(* CODESYS project codesys-syslog-library-history
   Author: John te Bokkel
   Company: PowerCore Engineering
   CompiledLibraryCompatibilityVersion: CODESYS V3.5 SP16
   DefaultNamespace: Syslog
   Description: Library project to implement RFC 5424 The Syslog Protocol
   DocFormat: reStructuredText
   LanguageModelAttribute: qualified-access-only
   Placeholder: CODESYS_SYSLOG
   Title: Code-Syslog
   Version: 0.1.0.0

Project tree, tasks and I/O mapping:
  libraries: CAA Types Extern, 3.5.17.0 (CAA Technical Workgroup); CAA FB Factory, 3.5.17.0 (CAA Technical Workgroup); Common Behaviour Model, 3.5.17.0 (3S - Smart Software Solutions GmbH); StringUtils, * (System); Code-Syslog Interfaces, * (PowerCore Engineering); SysTimeRtc, 3.5.17.0 (System); Element Collections, 3.5.17.0 (3S - Smart Software Solutions GmbH); CAA File, 3.5.17.0 (CAA Technical Workgroup); Net Base Services, 3.5.17.0 (3S - Smart Software Solutions GmbH); CmpIecTask, 3.5.17.0 (System); CmpCrypto, 3.5.17.0 (System); Standard, 3.5.18.0 (System)
  code-syslog/
  oscat-basic/
    function BIT_COUNT [ST]
    function D_TRUNC [ST]
    function FRACT [ST]
    function RDM [ST]
    function T_PLC_MS [ST]
  Handlers/
    Rotator/
    function block SyslogFileHandler [ST]: Dispatch, p_FlushNow, p_LogSeverity, prvFileSetup, prvFlush, prvProcessQueue, Run
    function block SyslogHandlerBase [ST]: Dispatch, p_LogSeverity, Run
    function block SyslogRotatingFileHandler [ST]: DoRollover, Rotate, RotationFilename, ShouldRollover
    function block SyslogRotatingFileHandlerBase [ST]: Run
    function block SyslogUdpHandler [ST]: prvInit, prvProcessQueue, prvSetupConnection, Run
  Syslog Msg Collection/
    function block IDataSyslogMsgElement [ST]
    interface ISyslogMsgElement: SyslogMsgValue
    function block SyslogMsgElement [ST]: ElementCompareTo, ElementEquals, ElementHashCode, prvInstInit, SyslogMsgValue
    function block SyslogMsgElementFactory [ST]: Create, prvInstCount, prvInstPoolExtendsFactor, prvInstSize
  function block SyslogLogger [ST]: FB_Init, Alert, Critical, Debug, Emergency, Error, Information, Notice, Warning, GetAppName, GetFacility, GetHostname, GetProcId, GetVersion, RegisterHandler, SetAppName, SetFacility, SetHostname, SetProcId, UnregisterHandler, prvBuildSyslogMessage, prvDispatch, prvTimestamp
  function Escape_ParamValue [ST]
  function Make_Priority [ST]
  function Make_SdParam2 [ST]
  function Make_SdParam [ST]
  function Make_SdParamSb [ST]
  function RandomEmpherialPort [ST]
  SafeLog/
    function SyslogAlert [ST]
    function SyslogCritical [ST]
    function SyslogDebug [ST]
    function SyslogEmergency [ST]
    function SyslogError [ST]
    function SyslogInfo [ST]
    function SyslogNotice [ST]
    function SyslogWarning [ST]
  function Sanitize_Msg [ST]
  function Sanitize_PrintUsAscii [ST]
  function Sanitize_SdName [ST]
  function StrucDataMsg [ST]
  function UtcTimestamp [ST]
  function UtcTimestampFromSystimeDate [ST]
  global variables Constants
*)

// Constants
{attribute 'qualified_only'}
//{attribute 'conditionalshow'}
//{attribute 'conditionalshow' := 'SomeText'}
//{attribute 'hide'}
VAR_GLOBAL CONSTANT
	gc_uiMaxHandlers : UINT := 5; /// Max number of registered log handlers
END_VAR

// Handlers/SyslogRotatingFileHandlerBase/DoRollover
/// Perform the rollover
/// :returns: TRUE when complete
{warning 'Add method implementation '}
METHOD PROTECTED DoRollover : BOOL
VAR_INPUT
END_VAR

// Handlers/SyslogRotatingFileHandlerBase/Rotate
/// When rotating, rotate the current log.
/// 
/// This should manage the file handle for the current log file. (ie. close it and reopen)
{warning 'Add method implementation '}
METHOD PROTECTED Rotate : BOOL
VAR_INPUT
	(* The source filename. This is normally the base filename, eg ``test.log``*)
	source	: STRING(255);
	(* The destination filename. This is normally what the source is rotated to, eg ``test.log.1``*)
	dest	: STRING(255);
END_VAR

// Handlers/SyslogRotatingFileHandlerBase/RotationFilename
/// Transformation file naming method.
/// 
/// default_name will be ``sFullFilename.#``
{warning 'Add method implementation '}
METHOD PROTECTED RotationFilename : CAA.FILENAME
VAR_INPUT
	default_name : CAA.FILENAME;
END_VAR

// Handlers/SyslogRotatingFileHandlerBase/ShouldRollover
{warning 'Add method implementation '}
/// Determine if we should rollover for this message. This needs to return in one call.
/// This method needs to look at the next message to be written to determine if rollover should occur.
METHOD PROTECTED ShouldRollover : BOOL
VAR_INPUT
END_VAR

// oscat-basic/BIT_COUNT
FUNCTION BIT_COUNT : INT
VAR_INPUT
	IN : DWORD;
END_VAR


(*
version 1.1	10 sep 2007
programmer 	hugo
tested by		tobias

BIT_COUNT counts the amount True of bits in a dword.
for exabple: bit_count(3) returns 2 because two bits (bits 0 and 1) are true and all others are false. 

*)

WHILE in > 0 DO
	IF in.0 THEN Bit_Count := Bit_Count + 1; END_IF;
	in := SHR(in,1);
END_WHILE;



(* revision history
5.7.2007	rev 1.0		original version

10.9.2007	rev 1.1		hm
	changed algorithm for better performace
	the execution time has reduced by a factor of 5
	deleted unused variable temp
*)

END_FUNCTION

// oscat-basic/D_TRUNC
FUNCTION D_TRUNC : DINT
VAR_INPUT
	X : REAL;
END_VAR

(*
version 1.2	10. mar. 2009
programmer 	hugo
tested by		oscat

d_trunc truncates a real to a dint 1.5 will be 1 and -1.5 will be -1
d_trunc is necessary because many systems do not offer a trunc to a dint
also real_to_dint will not deliver the same result on different systems

*)

D_TRUNC := REAL_TO_DINT(X);
IF X > 0.0 THEN
	IF DINT_TO_REAL(D_TRUNC) > X THEN D_TRUNC := D_TRUNC - 1; END_IF;
ELSE
	IF DINT_TO_REAL(D_TRUNC) < X THEN D_TRUNC := D_TRUNC + 1; END_IF;
END_IF;


(* for systems that support a dint truncation this routine can be replaced by trunc() *)


(* revision history
hm	21. mar. 2008	rev 1.0
	original version

hm	31. oct. 2008	rev 1.1
	optimized performance

hm	10. mar. 2009	rev 1.2
	real constants updated to new systax using dot
*)

END_FUNCTION

// oscat-basic/FRACT
/// this function returns the fraction of a real number
/// fract(3.14) = 0.14
FUNCTION FRACT : REAL
VAR_INPUT
	x : REAL;
END_VAR


(*
version 1.3	10. mar. 2009
programmer 	hugo
tested by		tobias

this function returns the fraction of a real number
fract(3.14) = 0.14

*)

IF ABS(x) < 2.0E9 THEN
	FRACT := x - DINT_TO_REAL(D_TRUNC(x));
ELSE
	FRACT := 0.0;
END_IF;

(* revision history
hm	4. aug 2006	rev 1.0
	original version

hm	11. mar 2008	rev 1.1
	added dint_to_real for compatibility reasons
	now returns 0 for number > 2e9
	changed input to x

hm	21. mar. 2008	rev 1.2
	use D_trunc instead of TRUNC for compatibility reasons

hm	10. mar. 2009	rev 1.3
	real constants updated to new systax using dot

*)

END_FUNCTION

// oscat-basic/RDM
(*this function calculates a pseudo random number
to generate the number it reads the sps timer and calculates a random number between 0 and 1:
in order to use rdm more then once within one sps cycle it need to be called with different seed numbers LAST.
*)
FUNCTION RDM : REAL
VAR_INPUT
	last : REAL;
END_VAR
VAR
	tn : DWORD;
	tc : INT;
END_VAR
VAR CONSTANT
	E : REAL := 	2.71828182845904523536028747135266249;		(* Euler constant e *)
END_VAR

(*
version 1.9	10. mar. 2009
programmer 	hugo
tested by		tobias

this function calculates a pseudo random number
to generate the number it reads the sps timer and calculates a random number between 0 and 1:
in order to use rdm more then once within one sps cycle it need to be called with different seed numbers LAST.

*)

tn := T_PLC_MS();
tc := BIT_COUNT(tn);
tn.31 := tn.2;
tn.30 := tn.5;
tn.29 := tn.4;
tn.28 := tn.1;
tn.27 := tn.0;
tn.26 := tn.7;
tn.25 := tn.6;
tn.24 := tn.3;
tn := ROL(tn,BIT_COUNT(tn)) OR 16#80000001;
tn := tn MOD 71474513 + INT_TO_DWORD(tc + 77);
RDM := FRACT(DWORD_TO_REAL(tn) / 10000000.0 * (E - LIMIT(0.0,last,1.0)));


(*
pt := ADR(temp);
pt^ := (T_PLC_MS() AND 16#007FFFFF) OR 16#3D000000;
RDM := fract(modR(temp*e+pi1, PI1-last) + modR(temp*PI1+e + last,e-last));
*)

(* revision history
hm		16. jan 2007		rev 1.0
	original version

hm		11. nov 2007		rev 1.1
	changed time() into t_plc_ms()

hm		20. nov 2007		rev 1.2
	changed code of temp calculation to avoid overflow in modr due to resuclt would not fit DINT for high timeer values

hm		5. jan 2008		rev 1.3
	changed calculation of temp to avoid problem with high values of t_plc_ms

hm		2. feb 2008		rev 1.4
	changed algorithm to avoind non iec functions and guarantee more randomness

hm	10. mar. 2008		rev 1.5
	make sure last will be between 0 and 1 to avoid invalid results

hm	16. mar. 2008		rev 1.6
	added conversion for tc to avoid warnings under codesys 3.0

hm	18. may. 2008		rev 1.7
	changed constant E to E1

hm	18. oct. 2008		rev 1.8
	using math constants

hm	10. mar. 2009		rev 1.9
	real constants updated to new systax using dot

*)

END_FUNCTION

// oscat-basic/T_PLC_MS
FUNCTION T_PLC_MS : DWORD
VAR CONSTANT
	debug : BOOL := 0;
	N : INT := 0;
	offset : DWORD := 0;
END_VAR
VAR
	tx : TIME;
END_VAR

(*
version 1.2	16. nov 2008
programmer 	hugo
tested by	oscat

T_PLC_MS reads the internal PLC timer and return the time, it has the advantage to be able to set a debug mode 
and speed up the counter to test the plc timer overrun which occurs every 50 days respectively 25 days at siemens S7
this routine also allows to correct the behavior of s7 where the internal plc counter will not count all 32 bits.

*)

tx := TIME();
T_PLC_MS := TIME_TO_DWORD(Tx);
(* hier muss die korrektur für step7 stattfinden
plctime muss den vollen wertebereich von time ausnutzen:
wenn bei step7 time -24tage bis plus 24 tage ist dann muss der timer auch beim überlauf auf -24tage springen 
und auf keinen fall auf 0 !!!!
für siemens muss ein weiterer fb im main eingebunden werden der sicherstellt das alle 32 bits durchgezählt werden.
es kann nur ein fb sein den er muss sich das oberste (32te) bit merken.
oder etwa spring s7 bei überlauf auf -24 tage????? dann wäre keine korrektur nötig.
*)
IF debug THEN
	T_PLC_MS := (SHL(T_PLC_MS,N) OR SHL(DWORD#1,N)-1) + OFFSET;
END_IF;

(* revision history
hm	14.9.2007	rev 1.0
	original version

hm	12. nov 2007	rev 1.1
	added temporaray variable tx because some compilers could not handle time() as an argument

hm	16. nov. 2008	rev 1.2
	initialized constants with 0 for compatibility reasons
*)

END_FUNCTION

// SyslogLogger
FUNCTION_BLOCK SyslogLogger IMPLEMENTS SyslogItfs.ISyslogLogger, SyslogItfs.ISyslogLoggerConfig
VAR_INPUT
END_VAR
VAR_OUTPUT
END_VAR
VAR
	_hostname : SyslogItfs.HOSTNAME := SyslogItfs.Constants.gc_sNILVALUE;
	_appName : SyslogItfs.APP_NAME := SyslogItfs.Constants.gc_sNILVALUE;
	_procId : SyslogItfs.PROC_ID := SyslogItfs.Constants.gc_sNILVALUE;
	_facility : SyslogItfs.SyslogFacility := SyslogItfs.SyslogFacility.USER;
	regHandler : ARRAY [0..c_iMaxHandler] OF SyslogItfs.ISyslogHandler;
	version : SyslogItfs.SYSLOG_VERSION := c_sVersion;
	ixHandler : INT;
END_VAR
VAR CONSTANT
	c_iMaxHandler : INT := UINT_TO_INT(Constants.gc_uiMaxHandlers) - 1;
	c_sVersion : STRING(2) := '1';
END_VAR

FOR ixHandler := 0 TO c_iMaxHandler BY 1 DO
	IF regHandler[ixHandler] <> CAA.gc_hINVALID THEN
		regHandler[ixHandler].Run();
	END_IF
END_FOR

//FB_Init is always available implicitly and it is used primarily for initialization.
//The return value is not evaluated. For a specific influence, you can also declare the
//methods explicitly and provide additional code there with the standard initialization
//code. You can evaluate the return value.
METHOD FB_Init: BOOL
VAR_INPUT
    bInitRetains: BOOL; // TRUE: the retain variables are initialized (reset warm / reset cold)
    bInCopyCode: BOOL;  // TRUE: the instance will be copied to the copy code afterward (online change)   
	hostname : SyslogItfs.HOSTNAME;
	appName : SyslogItfs.APP_NAME;
	procId : SyslogItfs.PROC_ID;
	facility : SyslogItfs.SyslogFacility;
	handler : SyslogItfs.ISyslogHandler;
END_VAR
THIS^._hostname := hostname;
THIS^._appName := appName;
THIS^._procId := procId;
THIS^._facility := facility;

THIS^.RegisterHandler(handler);
END_METHOD

METHOD Alert : BOOL
VAR_INPUT
	msgId	: SyslogItfs.MSG_ID;
	msg	: SyslogItfs.MSG;
END_VAR
THIS^.prvDispatch(SyslogItfs.SyslogSeverity.ALERT, ADR(msgId), ADR(msg));
END_METHOD

METHOD Critical : BOOL
VAR_INPUT
	msgId	: SyslogItfs.MSG_ID;
	msg	: SyslogItfs.MSG;
END_VAR
THIS^.prvDispatch(SyslogItfs.SyslogSeverity.CRITICAL, ADR(msgId), ADR(msg));
END_METHOD

METHOD Debug : BOOL
VAR_INPUT
	msgId	: SyslogItfs.MSG_ID;
	msg	: SyslogItfs.MSG;
END_VAR
THIS^.prvDispatch(SyslogItfs.SyslogSeverity.DEBUG, ADR(msgId), ADR(msg));
END_METHOD

METHOD Emergency : BOOL
VAR_INPUT
	msgId	: SyslogItfs.MSG_ID;
	msg	: SyslogItfs.MSG;
END_VAR
THIS^.prvDispatch(SyslogItfs.SyslogSeverity.EMERGENCY, ADR(msgId), ADR(msg));
END_METHOD


METHOD Error : BOOL
VAR_INPUT
	msgId	: SyslogItfs.MSG_ID;
	msg	: SyslogItfs.MSG;
END_VAR
THIS^.prvDispatch(SyslogItfs.SyslogSeverity.ERROR, ADR(msgId), ADR(msg));
END_METHOD


METHOD Information : BOOL
VAR_INPUT
	msgId	: SyslogItfs.MSG_ID;
	msg	: SyslogItfs.MSG;
END_VAR
THIS^.prvDispatch(SyslogItfs.SyslogSeverity.INFORMATION, ADR(msgId), ADR(msg));
END_METHOD


METHOD Notice : BOOL
VAR_INPUT
	msgId	: SyslogItfs.MSG_ID;
	msg	: SyslogItfs.MSG;
END_VAR
THIS^.prvDispatch(SyslogItfs.SyslogSeverity.NOTICE, ADR(msgId), ADR(msg));
END_METHOD


METHOD Warning : BOOL
VAR_INPUT
	msgId	: SyslogItfs.MSG_ID;
	msg	: SyslogItfs.MSG;
END_VAR
THIS^.prvDispatch(SyslogItfs.SyslogSeverity.WARNING, ADR(msgId), ADR(msg));
END_METHOD

METHOD GetAppName : SyslogItfs.APP_NAME
GetAppName := THIS^._appName;
END_METHOD

METHOD GetFacility : SyslogItfs.SyslogFacility
GetFacility := THIS^._facility;
END_METHOD

METHOD GetHostname : SyslogItfs.HOSTNAME
GetHostname := THIS^._hostname;
END_METHOD

METHOD GetProcId : SyslogItfs.PROC_ID
GetProcId := THIS^._procId;
END_METHOD

METHOD GetVersion : SyslogItfs.SYSLOG_VERSION
GetVersion := THIS^.version;
END_METHOD

/// Register Syslog Handler
/// :returns: TRUE if successfully added
METHOD RegisterHandler : BOOL
VAR_INPUT
	handler : SyslogItfs.ISyslogHandler;
END_VAR
VAR
	xDup : BOOL;
	ix : INT;
	ixOpen : INT;
END_VAR
IF handler <> CAA.gc_hINVALID THEN
	xDup := FALSE;
	ixOpen := -1;
	// We need to check the whole array for dups
	FOR ix := 0 TO c_iMaxHandler BY 1 DO
		xDup S= THIS^.regHandler[ix] = handler;
		IF ixOpen = -1 AND_THEN THIS^.regHandler[ix] = CAA.gc_hINVALID THEN
			ixOpen := ix;
		END_IF
	END_FOR
	
	IF NOT xDup THEN
		IF ixOpen >= 0 AND ixOpen <= c_iMaxHandler THEN
			THIS^.regHandler[ixOpen] := handler;
			RegisterHandler := TRUE;
		END_IF
	END_IF
END_IF
END_METHOD

(* Set App-Name According to RFC5424 Section 6.2.5*)
/// :returns: FALSE if we ended up with an empty/null string otherwise TRUE
METHOD SetAppName : BOOL
VAR_INPUT
	sAppName	: SyslogItfs.APP_NAME;
END_VAR
SetAppName := TRUE;
THIS^._appName := sAppName;

Sanitize_PrintUsAscii(ADR(THIS^._appName));
// Make sure we have a legal name after sanitizing it
IF stu.StrIsNullOrEmptyA(ADR(THIS^._appName)) THEN
	THIS^._appName := SyslogItfs.Constants.gc_sNILVALUE;
	SetAppName := FALSE;
END_IF
END_METHOD

METHOD SetFacility : SyslogItfs.SyslogFacility
VAR_INPUT
	facility	: SyslogItfs.SyslogFacility;
END_VAR
THIS^._facility := facility;
END_METHOD

(* Set the hostname according to RFC5424 Section 6.2.4*)
/// :returns: FALSE if we ended up with an empty/null string otherwise TRUE
METHOD SetHostname : BOOL
VAR_INPUT
	(* In order of preference FQDN, Static IP address, hostname, Dynamic IP address, NILVALUE*)
	sHostname	: SyslogItfs.HOSTNAME;
END_VAR
SetHostname := TRUE;
THIS^._hostname := sHostname;

Sanitize_PrintUsAscii(ADR(THIS^._hostname));
IF Stu.StrIsNullOrEmptyA(ADR(THIS^._hostname)) THEN
	THIS^._hostname := SyslogItfs.Constants.gc_sNILVALUE;
	SetHostname := FALSE;
END_IF
END_METHOD

(* Set Proc ID According to RFC 5424 Section 6.2.6*)
METHOD SetProcId : BOOL
VAR_INPUT
	sProcId	: SyslogItfs.PROC_ID;
END_VAR
SetProcId := TRUE;
THIS^._procId := sProcId;

Sanitize_PrintUsAscii(ADR(THIS^._procId));
IF Stu.StrIsNullOrEmptyA(ADR(THIS^._procId)) THEN
	THIS^._procId := SyslogItfs.Constants.gc_sNILVALUE;
	SetProcId := FALSE;
END_IF
END_METHOD

METHOD UnregisterHandler : BOOL
VAR_INPUT
	handler : SyslogItfs.ISyslogHandler;
END_VAR
VAR
	ix : INT;
END_VAR
IF handler <> CAA.gc_hINVALID THEN
	FOR ix := 0 TO c_iMaxHandler BY 1 DO
		IF THIS^.regHandler[ix] = handler THEN
			THIS^.regHandler[ix] := CAA.gc_hINVALID;
			UnregisterHandler := TRUE;
		END_IF
	END_FOR
END_IF
END_METHOD

METHOD PRIVATE prvBuildSyslogMessage : SyslogItfs.SYSLOG_MSG
VAR_INPUT
	severity : SyslogItfs.SyslogSeverity;
	pmsgId : POINTER TO SyslogItfs.MSG_ID;
	pmsg : POINTER TO SyslogItfs.MSG;
	ptimestamp : POINTER TO SyslogItfs.TIMESTAMP;
END_VAR
VAR
	pSysMsg : POINTER TO SyslogItfs.SYSLOG_MSG;
END_VAR
pSysMsg := ADR(prvBuildSyslogMessage);
// PRI VERSION SP
prvBuildSyslogMessage := concat(Make_Priority(severity, THIS^._facility), concat(THIS^.GetVersion(), SyslogItfs.gc_sSP));
// PRI VERSION SP TIMESTAMP
Stu.StrConcatA(ptimestamp, pSysMsg, UINT_TO_INT(SyslogItfs.gc_szSyslogMsg));
// PRI VERSION SP TIMESTAMP SP
Stu.StrConcatA(ADR(SyslogItfs.gc_sSP), pSysMsg, UINT_TO_INT(SyslogItfs.gc_szSyslogMsg));
// PRI VERSION SP TIMESTAMP SP HOSTNAME
Stu.StrConcatA(ADR(THIS^._hostname), pSysMsg, UINT_TO_INT(SyslogItfs.gc_szSyslogMsg));
// PRI VERSION SP TIMESTAMP SP HOSTNAME SP
Stu.StrConcatA(ADR(SyslogItfs.gc_sSP), pSysMsg, UINT_TO_INT(SyslogItfs.gc_szSyslogMsg));
// PRI VERSION SP TIMESTAMP SP HOSTNAME SP APP-NAME
Stu.StrConcatA(ADR(THIS^._appName), pSysMsg, UINT_TO_INT(SyslogItfs.gc_szSyslogMsg));
// PRI VERSION SP TIMESTAMP SP HOSTNAME SP APP-NAME SP
Stu.StrConcatA(ADR(SyslogItfs.gc_sSP), pSysMsg, UINT_TO_INT(SyslogItfs.gc_szSyslogMsg));
// PRI VERSION SP TIMESTAMP SP HOSTNAME SP APP-NAME SP PROCID
Stu.StrConcatA(ADR(THIS^._procId), pSysMsg, UINT_TO_INT(SyslogItfs.gc_szSyslogMsg));
// PRI VERSION SP TIMESTAMP SP HOSTNAME SP APP-NAME SP PROCID SP
Stu.StrConcatA(ADR(SyslogItfs.gc_sSP), pSysMsg, UINT_TO_INT(SyslogItfs.gc_szSyslogMsg));
// PRI VERSION SP TIMESTAMP SP HOSTNAME SP APP-NAME SP PROCID SP MSGID
Stu.StrConcatA(pmsgId, pSysMsg, UINT_TO_INT(SyslogItfs.gc_szSyslogMsg));
// HEADER SP
Stu.StrConcatA(ADR(SyslogItfs.gc_sSP), pSysMsg, UINT_TO_INT(SyslogItfs.gc_szSyslogMsg));
// HEADER SP MSG (the message part can contain both STRUCTURED-DATA and MSG)
Stu.StrConcatA(pmsg, pSysMsg, UINT_TO_INT(SyslogItfs.gc_szSyslogMsg));
END_METHOD

METHOD PRIVATE prvDispatch : BOOL
VAR_INPUT
	severity : SyslogItfs.SyslogSeverity;
	pmsgId : POINTER TO SyslogItfs.MSG_ID;
	pmsg : POINTER TO SyslogItfs.MSG;
END_VAR
VAR
	ix : INT;
	xTimestamp : BOOL;
	timestamp : SyslogItfs.TIMESTAMP;
END_VAR
FOR ix := 0 TO c_iMaxHandler BY 1 DO
	IF THIS^.regHandler[ix] <> CAA.gc_hINVALID THEN
		IF THIS^.regHandler[ix].p_LogSeverity >= severity THEN
			// We want all handlers to get the same timestamp
			IF NOT xTimestamp THEN
				timestamp := prvTimestamp();
				xTimestamp := TRUE;
			END_IF
			THIS^.regHandler[ix].Dispatch(THIS^.prvBuildSyslogMessage(severity, pmsgId, pmsg, ADR(timestamp)));
		END_IF
	END_IF
END_FOR
END_METHOD

/// prvTimestamp exists so we can override the timestamp for testing
METHOD PROTECTED prvTimestamp : SyslogItfs.TIMESTAMP
VAR_INPUT
END_VAR
prvTimestamp := UtcTimestamp();
END_METHOD

END_FUNCTION_BLOCK

// Sanitize_PrintUsAscii
/// Remove any non-printable ascii as defined by RFC5424
///
/// :return: TRUE if any characters removed.
FUNCTION Sanitize_PrintUsAscii : BOOL
VAR_INPUT
	// Pointer to String to sanitize
	cbpValue : Stu.CharBufferPtr;
END_VAR
VAR
	pChar : POINTER TO BYTE;
	pCursor : POINTER TO BYTE;
	iPos : UINT;
END_VAR

pChar := cbpValue;
pCursor := cbpValue;

WHILE pChar^ <> 0 DO
	// Copy current character to cursor position if it is valid printable ascii otherwise just advance to the next char
	IF (pChar^ < SyslogItfs.Constants.gc_byPRINTUSASCII_MIN OR pChar^ > SyslogItfs.Constants.gc_byPRINTUSASCII_MAX)
	THEN
		pChar := pChar + 1;
	ELSE
		pCursor^ := pChar^;
		pChar := pChar + 1;
		pCursor := pCursor + 1;
	END_IF
END_WHILE

// Null Terminate String at final cursor position
pCursor^ := 0;
// If we removed any characters return TRUE
Sanitize_PrintUsAscii := pChar <> pCursor;

END_FUNCTION

// Make_Priority
/// Make Priority string as per RFC5424 Section 6.2.1
FUNCTION Make_Priority : SyslogItfs.PRI
VAR_INPUT
	severity : SyslogItfs.SyslogSeverity;
	facility : SyslogItfs.SyslogFacility;
END_VAR
VAR
	prival : INT;
END_VAR

// bit shift facility by 3 the same as facility * 8 but faster
prival := SHL(TO_INT(facility), 3) + TO_INT(severity);
Make_Priority := concat('<', concat(INT_TO_STRING(prival), '>'));

END_FUNCTION

// UtcTimestamp
/// The current time as RFC5424 UTC TIMESTAMP
FUNCTION UtcTimestamp : SyslogItfs.TIMESTAMP
VAR_INPUT
END_VAR
VAR
	timestamp : SysTimeRtc.SYSTIME;
	rtsDate : SysTimeRtc.SYSTIMEDATE;
END_VAR

SysTimeRtc.SysTimeRtcHighResGet(timestamp);
SysTimeRtc.SysTimeRtcConvertHighResToDate(timestamp, rtsDate);
UtcTimestamp := UtcTimestampFromSystimeDate(rtsDate);

END_FUNCTION

// UtcTimestampFromSystimeDate
/// Convert a SysTimeRtc.SYSTIMEDATE object into a RFC5424 compliant UTC TIMESTAMP
FUNCTION UtcTimestampFromSystimeDate : SyslogItfs.TIMESTAMP
VAR_INPUT
	rtsDate : SysTimeRtc.SYSTIMEDATE;
END_VAR
VAR
	sf2d : STRING(5) := '%02d';
	sf3d : STRING(5) := '%03d';
	sf4d : STRING(5) := '%04d';
	sFormatted : STRING(10);
	psFormatted : POINTER TO STRING(10) := ADR(sFormatted);
	udiSize : UDINT := SIZEOF(sFormatted);
END_VAR

// Year
Stu.StuSprintf(ADR(sf4d), ADR(rtsDate.wYear), __SYSTEM.TYPE_CLASS.TYPE_UINT, psFormatted, udiSize);
UtcTimestampFromSystimeDate := concat(sFormatted, '-');

// Month
Stu.StuSprintf(ADR(sf2d), ADR(rtsDate.wMonth), __SYSTEM.TYPE_CLASS.TYPE_UINT, psFormatted, udiSize);
UtcTimestampFromSystimeDate := concat(UtcTimestampFromSystimeDate, concat(sFormatted, '-'));

// Day
Stu.StuSprintf(ADR(sf2d), ADR(rtsDate.wDay), __SYSTEM.TYPE_CLASS.TYPE_UINT, psFormatted, udiSize);
UtcTimestampFromSystimeDate := concat(UtcTimestampFromSystimeDate, concat(sFormatted, 'T'));

// Hour
Stu.StuSprintf(ADR(sf2d), ADR(rtsDate.wHour), __SYSTEM.TYPE_CLASS.TYPE_UINT, psFormatted, udiSize);
UtcTimestampFromSystimeDate := concat(UtcTimestampFromSystimeDate, concat(sFormatted, ':'));

// Minute
Stu.StuSprintf(ADR(sf2d), ADR(rtsDate.wMinute), __SYSTEM.TYPE_CLASS.TYPE_UINT, psFormatted, udiSize);
UtcTimestampFromSystimeDate := concat(UtcTimestampFromSystimeDate, concat(sFormatted, ':'));

// Second
Stu.StuSprintf(ADR(sf2d), ADR(rtsDate.wSecond), __SYSTEM.TYPE_CLASS.TYPE_UINT, psFormatted, udiSize);
UtcTimestampFromSystimeDate := concat(UtcTimestampFromSystimeDate, concat(sFormatted, '.'));

// Milli-Second
Stu.StuSprintf(ADR(sf3d), ADR(rtsDate.wMilliseconds), __SYSTEM.TYPE_CLASS.TYPE_UINT, psFormatted, udiSize);
UtcTimestampFromSystimeDate := concat(UtcTimestampFromSystimeDate, concat(sFormatted, 'Z'));

END_FUNCTION

// Escape_ParamValue
/// Escape Parameter Value.
/// 
/// If the character to escape is the last character in the buffer it will not be escaped as that would result in a buffer over-run 
///
/// :escape backslash: \\ (16#5c)
/// :escape right bracket: ] (16#5d)
/// :escape double quote: " (16#22)
/// :return: TRUE if any escape attempted
/// 
FUNCTION Escape_ParamValue : BOOL
VAR_INPUT
	// Pointer Paramater Value buffer
	pValue : POINTER TO SyslogItfs.PARAM_VALUE;
	// Value Buffer Size
	uiSize : UINT;
END_VAR
VAR
	pChar : POINTER TO BYTE;
	pNext : POINTER TO BYTE;
	iPos : INT;
	sReplacement : STRING(2) := '\\';
	pRep2nd : POINTER TO BYTE;
END_VAR
VAR CONSTANT
	BACKSLASH : BYTE := 92;
	RBRACKET : BYTE := 93;
	DQ : BYTE := 34;
END_VAR

pChar := pValue;
pNext := pChar + 1;
iPos := 1;
pRep2nd := ADR(sReplacement);
// Position of the character to escape
pRep2nd := pRep2nd + 1;
WHILE pChar^ <> 0 DO
	IF pChar^ = BACKSLASH AND NOT (pNext^ = BACKSLASH OR pNext^ = RBRACKET OR pNext^ = DQ) 
		OR pChar^ = RBRACKET
		OR pChar^ = DQ
	THEN
		// Found something to escape
		Escape_ParamValue := TRUE;
		pRep2nd^ := pChar^;
		Stu.StrReplaceA(pValue, uiSize, ADR(sReplacement), DINT_TO_INT(Stu.StrLenA(pValue)), 1, 2, iPos);
		// Advance 2 characters (passed the newly escaped value)
		pChar := pNext + 1;
		pNext := pChar + 1;
		iPos := DWORD_TO_INT(pNext - pValue);
		
	ELSE
		// If we are already escaped we move an additional char (total of 2)
		IF pChar^ = BACKSLASH AND (pNext^ = BACKSLASH OR pNext^ = RBRACKET OR pNext^ = DQ) THEN
			pChar := pChar + 1;
			pNext := pChar + 1;
		END_IF
		// Advance to next char
		pChar := pChar + 1;
		pNext := pChar + 1;
		iPos := DWORD_TO_INT(pNext - pValue);
	END_IF
	
	// Prevent buffer over run
	IF INT_TO_UINT(iPos) > uiSize THEN
		RETURN;
	END_IF
	
END_WHILE

END_FUNCTION

// Make_SdParam2
/// Make Structured Data Parameter
///
/// :returns: SD-PARAM        = PARAM-NAME "=" %d34 PARAM-VALUE %d34 example: uid="1234"
FUNCTION Make_SdParam2 : SyslogItfs.STRUCTURED_DATA
VAR_INPUT
	// Parameter name
	name : SyslogItfs.PARAM_NAME;
	// Value
	value : STRING(255);
END_VAR
VAR
END_VAR

Escape_ParamValue(ADR(value), SIZEOF(value));
Sanitize_SdName(ADR(name));
Make_SdParam2 := name;
Stu.StrConcatA(pstFrom:=ADR(SyslogItfs.gc_sEQ), pstTo:=ADR(Make_SdParam2), UINT_TO_INT(SyslogItfs.gc_szStructuredData));
Stu.StrConcatA(pstFrom:=ADR(SyslogItfs.gc_sDQ), pstTo:=ADR(Make_SdParam2), UINT_TO_INT(SyslogItfs.gc_szStructuredData));
Stu.StrConcatA(pstFrom:=ADR(value), pstTo:=ADR(Make_SdParam2), UINT_TO_INT(SyslogItfs.gc_szStructuredData));
Stu.StrConcatA(pstFrom:=ADR(SyslogItfs.gc_sDQ), pstTo:=ADR(Make_SdParam2), UINT_TO_INT(SyslogItfs.gc_szStructuredData));

END_FUNCTION

// Sanitize_SdName
/// Remove any non-printable ascii as defined by RFC5424 and any of the following
///
/// :remove equals: '=' (16#3d)
/// :remove right bracket: ']' (16#5d)
/// :remove space: ' ' (16#20)
/// :remove double quote: '"' (16#22)
///
/// :return: TRUE if any characters removed.
FUNCTION Sanitize_SdName : BOOL
VAR_INPUT
	// Pointer Structured Data Name buffer (string)
	psdName : POINTER TO SyslogItfs.SD_NAME;
END_VAR
VAR
	pChar : POINTER TO BYTE;
	pCursor : POINTER TO BYTE;
	iPos : UINT;
END_VAR

pChar := psdName;
pCursor := psdName;

WHILE pChar^ <> 0 DO
	// Copy current character to cursor position if it is valid printable ascii otherwise just advance to the next char
	IF (pChar^ < SyslogItfs.Constants.gc_byPRINTUSASCII_MIN OR pChar^ > SyslogItfs.Constants.gc_byPRINTUSASCII_MAX)
		OR pChar^ = SyslogItfs.Constants.gc_bySP
		OR pChar^ = 61 // '='
		OR pChar^ = 93 // ']'
		OR pChar^ = 34 // '"'
	THEN
		pChar := pChar + 1;
	ELSE
		pCursor^ := pChar^;
		pChar := pChar + 1;
		pCursor := pCursor + 1;
	END_IF
END_WHILE

// Null Terminate String at final cursor position
pCursor^ := 0;
// If we removed any characters return TRUE
Sanitize_SdName := pChar <> pCursor;

END_FUNCTION

// Make_SdParam
/// Make Structured Data Parameter
///
/// :returns: SD-PARAM        = PARAM-NAME "=" %d34 PARAM-VALUE %d34 example: uid="1234"
FUNCTION Make_SdParam : SyslogItfs.STRUCTURED_DATA
VAR_INPUT
	// Parameter Name
	name : SyslogItfs.PARAM_NAME;
	// Pointer to Paramater value
	value : SyslogItfs.PARAM_VALUE;
	// Size of Value buffer
	szValue : UINT;
END_VAR
VAR
END_VAR

Escape_ParamValue(value, szValue);
Sanitize_SdName(ADR(name));
Make_SdParam := name;
Stu.StrConcatA(pstFrom:=ADR(SyslogItfs.gc_sEQ), pstTo:=ADR(Make_SdParam), UINT_TO_INT(SyslogItfs.gc_szStructuredData));
Stu.StrConcatA(pstFrom:=ADR(SyslogItfs.gc_sDQ), pstTo:=ADR(Make_SdParam), UINT_TO_INT(SyslogItfs.gc_szStructuredData));
Stu.StrConcatA(pstFrom:=value, pstTo:=ADR(Make_SdParam), UINT_TO_INT(SyslogItfs.gc_szStructuredData));
Stu.StrConcatA(pstFrom:=ADR(SyslogItfs.gc_sDQ), pstTo:=ADR(Make_SdParam), UINT_TO_INT(SyslogItfs.gc_szStructuredData));

END_FUNCTION

// Make_SdParamSb
/// Make Structured Data Parameter
///
/// :returns: UINT Number of characters appended        = PARAM-NAME "=" %d34 PARAM-VALUE %d34 example: uid="1234"
FUNCTION Make_SdParamSb : UINT
VAR_INPUT
	sb : PSBItfs.IStringBuilder;
	// Parameter name
	name : SyslogItfs.PARAM_NAME;
	// Value
	value : STRING(255);
END_VAR
VAR
	uiStart : UINT;
END_VAR

IF sb <> 0 THEN
	{IF (hastype (variable: sb.p_length, __UXINT))}
	uiStart := __UXINT_TO_UINT(sb.p_length);
	{ELSE}
	uiStart := UDINT_TO_UINT(sb.p_length);
	{END_IF}
	
	Escape_ParamValue(ADR(value), SIZEOF(value));
	Sanitize_SdName(ADR(name));
	
	sb.Append(name);
	sb.Append(SyslogItfs.gc_sEQ);
	sb.Append(SyslogItfs.gc_sDQ);
	sb.Append(value);
	sb.Append(SyslogItfs.gc_sDQ);
	
	{IF (hastype (variable: sb.p_length, __UXINT))}
	Make_SdParamSb := __UXINT_TO_UINT(sb.p_length) - uiStart;
	{ELSE}
	Make_SdParamSb := UDINT_TO_UINT(sb.p_length) - uiStart;
	{END_IF}
ELSE
	Make_SdParamSb := 0;
END_IF

END_FUNCTION

// RandomEmpherialPort
FUNCTION RandomEmpherialPort : UINT
VAR_INPUT
END_VAR
VAR
	dwRandBytes : DWORD;
	rand : REAL;
	eError : CmpCrypto_Interfaces.RTS_IEC_RESULT;
	abyRand : ARRAY [0..3] OF BYTE;
	rbs : CmpCrypto_Interfaces.RtsByteString;
END_VAR
VAR CONSTANT
	rfcLow : UINT := 49152;
	rfcHigh : UINT := 65535;
END_VAR

eError := CmpCrypto_Implementation.CryptoRtsByteStringInit2(ADR(rbs), 4, ADR(abyRand), FALSE);
eError := CmpCrypto_Implementation.CryptoGenerateRandomNumber(4, ADR(rbs));
dwRandBytes := SHL(BYTE_TO_DWORD(abyRand[0]), 24) OR SHL(BYTE_TO_DWORD(abyRand[1]), 16) OR SHL(BYTE_TO_DWORD(abyRand[2]), 8) OR BYTE_TO_DWORD(abyRand[3]); 

// divide dword by max dword to get a REAL fractional number <= 1.0
rand := DWORD_TO_REAL(dwRandBytes) / 16#FFFFFFFF;
RandomEmpherialPort := INT_TO_UINT(TRUNC_INT(rand * UINT_TO_REAL(rfcHigh - rfcLow + 1))) + rfcLow;

END_FUNCTION

// Sanitize_Msg
/// Sanitize Message according to RFC5424.
///
/// Control characters are replaced with as escaped hex strings
/// 
/// 6.4.  MSG
/// ^^^^^^^^^
/// 
///    The MSG part contains a free-form message that provides information
///    about the event.
/// 
///    The character set used in MSG SHOULD be UNICODE, encoded using UTF-8
///    as specified in [RFC3629].  If the syslog application cannot encode
///    the MSG in Unicode, it MAY use any other encoding.
/// 
///    The syslog application SHOULD avoid octet values below 32 (the
///    traditional US-ASCII control character range except DEL).  These
///    values are legal, but a syslog application MAY modify these
///    characters upon reception.  For example, it might change them into an
///    escape sequence (e.g., value 0 may be changed to "\\0").  A syslog
///    application SHOULD NOT modify any other octet values.
/// 
///    If a syslog application encodes MSG in UTF-8, the string MUST start
///    with the Unicode byte order mask (BOM), which for UTF-8 is ABNF
///    %xEF.BB.BF.  The syslog application MUST encode in the "shortest
///    form" and MAY use any valid UTF-8 sequence.
/// 
/// :return: TRUE if any changes occur.
/// 

FUNCTION Sanitize_Msg : BOOL
VAR_INPUT
	// Pointer to String to sanitize
	cbpValue : Stu.CharBufferPtr;
	// Size of cbpValue buffer
	uiSize : UINT;
END_VAR
VAR
	control : BYTE;
	// Initialized because for some reason trying to write to the first byte
	// of a zero length string doesn't work, but if it has length it does.
	sControl : STRING(2) := 'a';
	psControl : POINTER TO BYTE := ADR(sControl);
	sEscapeFormat : STRING(8) := '\x%02x';
	sEscape : STRING(8);
	iPos : INT;
END_VAR

// Escape all control characters as hex string escapes
// 10#31 becomes '\x1f' and 10#8 becomes '\x08'
FOR control := 1 TO 31 BY 1 DO
	psControl^ := control;
	Stu.StuSprintf(ADR(sEscapeFormat), ADR(control), __SYSTEM.TYPE_CLASS.TYPE_BYTE, ADR(sEscape), SIZEOF(sEscape));
	iPos := Stu.StrFindA(cbpValue, psControl, 0);
	WHILE iPos > 0 DO
		Sanitize_Msg := TRUE;
		Stu.StrReplaceA(cbpValue, uiSize, ADR(sEscape), DINT_TO_INT(Stu.StrLenA(cbpValue)), 1, DINT_TO_INT(Stu.StrLenA(ADR(sEscape))), iPos);
		iPos := Stu.StrFindA(cbpValue, psControl, INT_TO_UINT(iPos + 1));
	END_WHILE
END_FOR

END_FUNCTION

// StrucDataMsg
FUNCTION StrucDataMsg : SyslogItfs.MSG
VAR_INPUT
	itfStructData : SyslogItfs.IStructuredData;
	msg : SyslogItfs.MSG;
END_VAR
VAR
	lenSd : DINT;
	lenMsg : DINT;
	pMsg : POINTER TO ARRAY [1..SyslogItfs.gc_szMsg] OF BYTE;
END_VAR

StrucDataMsg := itfStructData.AsStructuredData();
Stu.StrConcatA(pstFrom:=ADR(SyslogItfs.gc_sSP), pstTo:=ADR(StrucDataMsg), UINT_TO_INT(SIZEOF(StrucDataMsg)));
lenSd := Stu.StrLenA(ADR(StrucDataMsg));

Sanitize_Msg(ADR(msg), SIZEOF(msg));
lenMsg := Stu.StrLenA(ADR(msg));

IF (lenSd + lenMsg) > SIZEOF(StrucDataMsg) THEN
	pMsg := ADR(msg);
	// Truncate msg
	pMsg^[lenMsg + (SyslogItfs.gc_szMsg - lenSd - lenMsg + 1)] := 0;
END_IF

Stu.StrConcatA(pstFrom:=ADR(msg), pstTo:=ADR(StrucDataMsg), UINT_TO_INT(SIZEOF(StrucDataMsg)));

END_FUNCTION

// Handlers/SyslogFileHandler
{attribute 'reflection'}
FUNCTION_BLOCK SyslogFileHandler EXTENDS SyslogHandlerBase IMPLEMENTS SyslogItfs.ISyslogHandler
VAR_INPUT
	filename : CAA.FILENAME;
END_VAR
VAR_OUTPUT
END_VAR
VAR
	
	defaultDir : CAA.FILENAME := 'csyslog/';
	{attribute 'instance-path'}
	{attribute 'noinit'}
	sInstance: STRING(100);
	
	mxHandler : UINT;
	// File Setup
	hActiveFile : CAA.HANDLE;
	mxFileSetup : UINT;
	getPos : FILE.GetPos;
	fileExists : FILE.GetSize;
	szFilesize : UDINT;
	sFullFilename : CAA.FILENAME;

	// auto-flush timer
	tmrFlush : TON := (PT:=T#5M);
	// flush request
	xFlushNow : BOOL;
	// Queue idle
	xQueueBusy : BOOL;
END_VAR
VAR CONSTANT
	sEOL : STRING(2) := '$n';
END_VAR

METHOD Dispatch : BOOL
VAR_INPUT
	syslogMsg	: SyslogItfs.SYSLOG_MSG;
END_VAR
IF xDiscardOldMsgWhenQueueFull THEN
	// queue is full
	IF THIS^.queue.CountElements() >= THIS^.queue.udiMaxElements THEN
		// remove an element and just discard it
		THIS^.queue.Poll();
	END_IF
END_IF

IF NOT xError THEN
	THIS^.queue.AddElement(itfElement:=THIS^.SyslogMsgFactor.Create(ADR(syslogMsg)));
END_IF
END_METHOD

/// Flush file buffer to disk now
{attribute 'monitoring' := 'call'}
PROPERTY p_FlushNow : BOOL
GET
p_FlushNow := THIS^.xFlushNow;
END_GET
SET
THIS^.xFlushNow := p_FlushNow;
END_SET
END_PROPERTY

{attribute 'monitoring' := 'call'}
PROPERTY p_LogSeverity : SyslogItfs.SyslogSeverity
GET
p_LogSeverity := THIS^.severity;
END_GET
SET
THIS^.severity := p_LogSeverity;
END_SET
END_PROPERTY

METHOD PROTECTED prvFileSetup : BOOL
VAR_INPUT
END_VAR
VAR_INST
	lastError : FILE.ERROR;
	mkdir : FILE.DirCreate;
	open : FILE.Open;
	close : FILE.Close;

	openMode : FILE.MODE := FILE.MODE.MAPPD;
END_VAR
CASE mxFileSetup OF
	0: // Try and create our directory
		mkdir(xExecute:=TRUE, sDirName:=THIS^.defaultDir);
		IF mkdir.xError OR mkdir.xDone THEN
			IF mkdir.eError = FILE.ERROR.EXIST or mkdir.eError = FILE.ERROR.NO_ERROR THEN
				mxFileSetup := 10;
			ELSE
				mxFileSetup := 3000;
				lastError := mkdir.eError;
				xError := TRUE;
			END_IF
			
			IF mkdir.xDone THEN
				mxFileSetup := 10;
			END_IF
			mkdir(xExecute:=FALSE);
		END_IF
	10: // Filename setup
		IF NOT Stu.StrIsNullOrEmptyA(ADR(THIS^.filename)) THEN
			// if there are any directories in the path we use it as is
			IF find(THIS^.filename, '/') > 0 OR find(THIS^.filename, '\') > 0 THEN
				sFullFilename := THIS^.filename;
			ELSE
				// otherwise it goes in the default directory
				sFullFilename := concat(THIS^.defaultDir, THIS^.filename);
			END_IF
		ELSE
			// an unset filename will instead use the instance a filename
			sFullFilename := concat(THIS^.defaultDir, concat(THIS^.sInstance, '.log'));
		END_IF
		mxFileSetup := 15;
	15: // Close handle if still open
		IF hActiveFile <> CAA.gc_hINVALID THEN
			close(xExecute:=TRUE, hFile:=hActiveFile);
			IF close.xDone OR close.xError THEN
				IF close.xError THEN
					lastError := close.eError;
				END_IF
				hActiveFile := CAA.gc_hINVALID;
				close(xExecute:=FALSE);
				mxFileSetup := 20;
			END_IF
		ELSE
			mxFileSetup := 20;
		END_IF
	20: // Try to Open the file in append mode or fall back to normal write if file doesn't exist
		open(xExecute:=TRUE, sFileName:=sFullFilename, eFileMode:=openMode);
		IF open.xError OR open.xDone THEN
			IF open.xError THEN
				hActiveFile := CAA.gc_hINVALID;
				lastError := open.eError;
				IF open.eError = FILE.ERROR.NOT_EXIST THEN
					openMode := FILE.MODE.MWRITE;
				ELSE
					mxFileSetup := 5000;
				END_IF
			END_IF
			
			IF open.xDone THEN
				hActiveFile := open.hFile;
				openMode := FILE.MODE.MAPPD;
				mxFileSetup := 30;
			END_IF
			open(xExecute:=FALSE);
		END_IF
	30: // Check file size (via current position)
		getPos(xExecute:=TRUE, hFile:=hActiveFile);
		IF getPos.xDone OR getPos.xError THEN
			IF getPos.xError THEN
				xError := TRUE;
				mxFileSetup := 6000;
			ELSE
				mxFileSetup := 0;
				szFilesize := __UXINT_TO_UDINT(getPos.udiPos);
				prvFileSetup := TRUE;
			END_IF
			getPos(xExecute:=FALSE);
		END_IF
	ELSE
		prvFileSetup := FALSE;
		xDiscardOldMsgWhenQueueFull := TRUE;
END_CASE
END_METHOD

/// Flush file buffer to disk.
/// :returns: TRUE on done or error
METHOD PROTECTED prvFlush : BOOL
VAR_INPUT
END_VAR
VAR_INST
	flush : FILE.Flush;
END_VAR
flush(xExecute:=TRUE, hFile:=hActiveFile);
IF flush.xDone OR flush.xError THEN
	xError S= flush.xError;
	flush(xExecute:=FALSE);
	prvFlush := TRUE;
END_IF
END_METHOD

METHOD PROTECTED prvProcessQueue : BOOL
VAR_INPUT
END_VAR
VAR_INST
	sCurrentMsg : SyslogItfs.SYSLOG_MSG;
	write : FILE.Write;
	lastError : FILE.ERROR;
	tickStart : CAA.TICK;
	tickEnd : CAA.TICK;
END_VAR
VAR
	szLength : DINT;
END_VAR
CASE mxQueue OF
	0: // Idle
		xQueueBusy := FALSE;
		IF queue.CountElements() > 0 THEN
			xQueueBusy := TRUE;
			mxQueue := 10;
		END_IF
	10: // Get Element
		eError := queue.Poll(itfElement => THIS^.itfElement);
		IF __QUERYINTERFACE(itfElement, itfSyslogMsgElement) THEN
			sCurrentMsg := itfSyslogMsgElement.SyslogMsgValue;
			Stu.StrConcatA(pstFrom:=ADR(sEOL), pstTo:=ADR(sCurrentMsg), UINT_TO_INT(SIZEOF(sCurrentMsg)));
		END_IF
		
		IF eError = COL.COLLECTION_ERROR.NO_ERROR THEN
			mxQueue := 20;
		ELSE
			mxQueue := 0;
		END_IF
	20: // get size
		fileExists(xExecute:=TRUE, sFileName:=sFullFilename);
		IF fileExists.xDone OR fileExists.xError THEN
			tickEnd := FILE.TICKS.GetTick(TRUE);
			mxQueue := 30;
			IF fileExists.xError THEN
				lastError := fileExists.eError;
				mxQueue := 40;
			END_IF
			fileExists(xExecute:=FALSE);
		END_IF
	30: // write to file
		szLength := Stu.StrLenA(ADR(sCurrentMsg));
		write(xExecute:=TRUE, hFile:=THIS^.hActiveFile, pBuffer:=ADR(sCurrentMsg), szSize:=DINT_TO_UDINT(szLength));
		IF write.xDone OR write.xError THEN
			mxQueue := 0;
			IF write.xError THEN
				lastError := write.eError;
				xError := TRUE;
				mxQueue := 40;
			ELSE
				szFilesize := szFilesize + DINT_TO_UDINT(szLength);
			END_IF
			write(xExecute:=FALSE);
		END_IF

	40: // Handle write error
		CASE lastError OF
			FILE.ERROR.WRONG_PARAMETER,
			FILE.ERROR.ABORT:
				xError := TRUE;
			ELSE
				// Setting the main loop back to init
				mxHandler := 0;
				// come back to trying to write the last message to file
				mxQueue := 20;
		END_CASE
	ELSE
		; // NOP
END_CASE
END_METHOD

/// Run the handler
METHOD Run : BOOL
VAR_INPUT
END_VAR
IF NOT xError THEN
	
	CASE mxHandler OF
		0: // Init
			IF prvFileSetup() THEN
				mxHandler := 10;
			END_IF
		10: // Process Queue
			prvProcessQueue();
			tmrFlush(IN:=TRUE);
			IF tmrFlush.Q OR xFlushNow THEN
				IF prvFlush() THEN
					tmrFlush(IN:=FALSE);
					xFlushNow := FALSE;
				END_IF
			END_IF
		20: // Reset?
			mxHandler := 0;
	END_CASE
	
END_IF
END_METHOD

END_FUNCTION_BLOCK

// Handlers/SyslogHandlerBase
FUNCTION_BLOCK SyslogHandlerBase IMPLEMENTS SyslogItfs.ISyslogHandler
VAR_INPUT
	severity : SyslogItfs.SyslogSeverity := SyslogItfs.SyslogSeverity.ERROR;
END_VAR
VAR_OUTPUT
	xError : BOOL;
END_VAR
VAR
	xDiscardOldMsgWhenQueueFull : BOOL;
	// Queue Processing
	mxQueue : UINT;
	aElements : ARRAY[0..999] OF COL.IElement; // Create an array of IElements for a static queue. NOTE: The size must be 2 times larger than the maximum number of used elements. 
	queue : COL.Queue := (paElements := ADR(aElements), udiMaxElements := 1000); // Created a static queue. NOTE: Static created elements of this queue will be online change safe.
	SyslogMsgFactor : SyslogMsgElementFactory;
	itfElement : COL.IElement;
	itfSyslogMsgElement : ISyslogMsgElement;
	eError : COL.COLLECTION_ERROR;
END_VAR

METHOD Dispatch : BOOL
VAR_INPUT
	syslogMsg	: SyslogItfs.SYSLOG_MSG;
END_VAR
IF xDiscardOldMsgWhenQueueFull THEN
	// queue is full
	IF THIS^.queue.CountElements() >= THIS^.queue.udiMaxElements THEN
		// remove an element and just discard it
		THIS^.queue.Poll();
	END_IF
END_IF


THIS^.queue.AddElement(itfElement:=THIS^.SyslogMsgFactor.Create(ADR(syslogMsg)));
Dispatch := TRUE;
END_METHOD

{attribute 'monitoring' := 'call'}
PROPERTY p_LogSeverity : SyslogItfs.SyslogSeverity
GET
p_LogSeverity := THIS^.severity;
END_GET
SET
THIS^.severity := p_LogSeverity;
END_SET
END_PROPERTY

(* Run the handler base code*)
METHOD Run : BOOL
END_METHOD

END_FUNCTION_BLOCK

// Syslog Msg Collection/SyslogMsgElementFactory
{attribute 'enable_dynamic_creation'}
FUNCTION_BLOCK SyslogMsgElementFactory EXTENDS COL.FBF.FactoryBase
VAR_INPUT
END_VAR
VAR_OUTPUT
END_VAR
VAR
END_VAR

SUPER^();

METHOD Create : ISyslogMsgElement
VAR_INPUT
	pmsg : POINTER TO SyslogItfs.SYSLOG_MSG;
END_VAR
VAR_OUTPUT
	eError : COL.FBF.ERROR;
END_VAR
VAR
	hInst : COL.CAA.HANDLE;
	itfInst : COL.FBF.IInstance;
	xOk : BOOL;
	itfData : IDataSyslogMsgElement;
	pInstance : POINTER TO SyslogMsgElement;
END_VAR
(* !!! This code must not be subject to change !!! *)
itfData(sValue := pmsg^);
hInst := SUPER^.prvAllocInstMem(eError => eError);
pInstance := SUPER^.prvGetInstPointer(hInst);
IF pInstance <> 0 AND eError = COL.FBF.ERROR.NO_ERROR THEN


	{implicit on}
	// This isn't actually an error
	pInstance^.__vfInit();
	pInstance^.FB_Init(TRUE, FALSE);
	{implicit off}


	xOk := __QUERYINTERFACE(pInstance^, itfInst);
	IF xOk THEN
		xOk := SUPER^.prvInstInit(itfInst, hInst, itfData, eError=>eError);
	ELSE
		eError := COL.FBF.ERROR.WRONG_INTERFACE;
	END_IF

	IF NOT xOk THEN
		SUPER^.prvFreeInstMem(hInst);
		Create := COL.CAA.gc_pNULL;
    ELSE
        __QUERYINTERFACE(pInstance^, Create);
	END_IF
END_IF
END_METHOD

/// Initial size of the heap alloc in number of instances
(* Is called by ``prvMemAlloc``, if ``prvPoolAdr`` returns ``CAA.gc_pNULL``*)
PROPERTY prvInstCount : FBF.CAA.COUNT
GET
// ~2048 * 10 = ~20KiB of heap to start with
prvInstCount := 10;
END_GET
END_PROPERTY

(* Is called by ``prvMemAlloc``, to determine the amout of memory growing (``MBM.PoolExtendH``)*)
PROPERTY prvInstPoolExtendsFactor : USINT
GET
(* This value will be interpreted as a 0..x% size extendsion related to the original size of the pool *)
prvInstPoolExtendsFactor := 10;
END_GET
END_PROPERTY

(* Is called by ``prvMemAlloc``. Should Implemented like :code:`prvInstSize := sizeof(CustomFB)`*)
PROPERTY prvInstSize : FBF.CAA.SIZE
GET
prvInstSize := sizeof(SyslogMsgElement);
END_GET
END_PROPERTY

END_FUNCTION_BLOCK

// Syslog Msg Collection/ISyslogMsgElement
INTERFACE ISyslogMsgElement EXTENDS COL.IElement

PROPERTY SyslogMsgValue : SyslogItfs.SYSLOG_MSG
GET
END_GET
END_PROPERTY

END_INTERFACE

// Syslog Msg Collection/IDataSyslogMsgElement
{attribute 'enable_dynamic_creation'}
{attribute 'hide'}
FUNCTION_BLOCK IDataSyslogMsgElement EXTENDS COL.FBF.InstanceData
VAR_INPUT
	sValue : SyslogItfs.SYSLOG_MSG;
END_VAR
VAR_OUTPUT
END_VAR
VAR
END_VAR

(* !! Do not add any executable code here !! *)
SUPER^();

END_FUNCTION_BLOCK

// Syslog Msg Collection/SyslogMsgElement
{attribute 'no_explicit_call' := 'Explicit calls not allowed.'}
FUNCTION_BLOCK SyslogMsgElement EXTENDS COL.FBF.InstanceBase IMPLEMENTS ISyslogMsgElement
VAR_INPUT
END_VAR
VAR_OUTPUT
END_VAR
VAR
	sSyslogMsg : SyslogItfs.SYSLOG_MSG;
END_VAR

(* Compares this element with itfElement.
 Returns 0 if the elements are equal, < 0 if the element is less than itfElement, 
 > 0 if the element is greater than itfElement.
 This method will be called from sorted collections (e.g. |SortedList|) to sort elements.
 IMPORTANT: The underlying value to be compared with MUST NOT be changed during the lifecycle of the object.*)
METHOD ElementCompareTo : INT
VAR_INPUT
	(* The element to compare*)
	itfElement	: COL.IElement;
END_VAR
VAR
	itfSyslogMsgElement : ISyslogMsgElement;
	sOther : SyslogItfs.SYSLOG_MSG;
END_VAR
IF __QUERYINTERFACE(itfElement, itfSyslogMsgElement) THEN
	sOther := itfSyslogMsgElement.SyslogMsgValue;
	ElementCompareTo := Stu.StrCmpA(ADR(THIS^.sSyslogMsg), ADR(sOther));
ELSE
	ElementCompareTo := -1;
END_IF
END_METHOD

(* Returns true of this element and itfElement are equal.
 This method will be called from the function block |HashTable| to find an element by key if the hashcode of an element collides with an other element.
 IMPORTANT: The underlying value to be compared with MUST NOT be changed during the lifecycle of the object.*)
METHOD ElementEquals : BOOL
VAR_INPUT
	(* The element to compare*)
	itfElement	: COL.IElement;
END_VAR
VAR
	itfSyslogMsgElement : ISyslogMsgElement;
	sOther : SyslogItfs.SYSLOG_MSG;
END_VAR
IF __QUERYINTERFACE(itfElement, itfSyslogMsgElement) THEN
	sOther := itfSyslogMsgElement.SyslogMsgValue;
	ElementEquals := Stu.StrCmpA(ADR(THIS^.sSyslogMsg), ADR(sOther)) = 0;
ELSE
	ElementEquals := FALSE;
END_IF
END_METHOD

(* Returns the hashcode of this element.
 This method is used by hash based collections (e.g. |Hashtable|) to get the hashcode from a element.
 IMPORTANT: The value of the method MUST NOT be changed during the lifecycle of the object.*)
METHOD ElementHashCode : LINT
// use the pointer address value as the hash
{warning disable C0196}
{warning disable C0033}
ElementHashCode := THIS;
{warning enable C0033}
{warning enable C0196}
END_METHOD

METHOD prvInstInit : FBF.ERROR (* eError *)
VAR_INPUT
	itfData	: FBF.IData;
END_VAR
VAR
	pData : POINTER TO IDataSyslogMsgElement;
END_VAR
SUPER^.prvInstInit(itfData);
IF __QUERYPOINTER(itfData, pData) THEN
	THIS^.sSyslogMsg := pData^.sValue;
END_IF
END_METHOD

PROPERTY SyslogMsgValue : SyslogItfs.SYSLOG_MSG
GET
SyslogMsgValue := THIS^.sSyslogMsg;
END_GET
END_PROPERTY

END_FUNCTION_BLOCK

// Handlers/SyslogRotatingFileHandler
FUNCTION_BLOCK SyslogRotatingFileHandler EXTENDS SyslogRotatingFileHandlerBase
VAR_INPUT
	// 1024^2 * 10 == 5120 lines @ gc_szSyslogMsg
	// This equates to 10 MiB
	szMaxFilesize : CAA.SIZE := 1048576;
	// backup count
	uiBackupCount : UINT := 5;
END_VAR
VAR_OUTPUT
END_VAR
VAR
END_VAR

(* Perform the rollover
 :returns: TRUE when complete*)
METHOD PROTECTED DoRollover : BOOL
VAR_INST
	ix : INT;
	mxRoll : UINT;
	sSource : CAA.FILENAME;
	sDest : CAA.FILENAME;
	rm : FILE.Delete;
	mv : FILE.Rename;
END_VAR
IF uiBackupCount > 0 THEN
	CASE mxRoll OF
		0: // Init
			// We go through the files in reverse
			ix := UINT_TO_INT(uiBackupCount) - 1;
			mxRoll := 10;
		10:
			sSource := concat(THIS^.sFullFilename, concat('.', INT_TO_STRING(ix)));
			sDest := concat(THIS^.sFullFilename, concat('.', INT_TO_STRING(ix + 1)));
			mxRoll := 20;
		20: // Remove dest
			rm(xExecute:=TRUE, sFileName:=sDest);
			IF rm.xDone OR rm.xError THEN
				rm(xExecute:=FALSE);
				IF ix < 1 THEN
					mxRoll := 40;
				ELSE
					ix := ix - 1;
					mxRoll := 30;
				END_IF
			END_IF
		30: // Move source to dest
			mv(xExecute:=TRUE, sFileNameOld:=sSource, sFileNameNew:=sDest);
			IF mv.xDone OR mv.xError THEN
				mv(xExecute:=FALSE);
				mxRoll := 10;
			END_IF
		40: // Rotate active log out
			IF THIS^.Rotate(THIS^.sFullFilename, sDest) THEN
				mxRoll := 0;
				DoRollover := TRUE;
			END_IF
	END_CASE
ELSE
	DoRollover := TRUE;
END_IF
END_METHOD

(* When rotating, rotate the current log.
 
 This should manage the file handle for the current log file. (ie. close it and reopen)*)
METHOD PROTECTED Rotate : BOOL
VAR_INPUT
	(* The source filename. This is normally the base filename, eg ``test.log``*)
	source	: STRING(255);
	(* The destination filename. This is normally what the source is rotated to, eg ``test.log.1``*)
	dest	: STRING(255);
END_VAR
VAR_INST
	mv : FILE.Rename;
	flush : FILE.Flush;
	close : FILE.Close;
	open : FILE.Open;
	mxRot : UINT;
	mxClose : UINT;
END_VAR
// We need to check if our pointer is valid AND if what it points to is a valid handle
IF hActiveFile <> CAA.gc_hINVALID THEN
	CASE mxClose OF
		0: // Flush
			flush(xExecute:=TRUE, hFile:=hActiveFile);
			IF flush.xDone OR flush.xError THEN
				flush(xExecute:=FALSE);
				mxClose := 10;
			END_IF
		10: // Close
			close(xExecute:=TRUE, hFile:=THIS^.hActiveFile);
			IF close.xDone OR close.xError THEN
				THIS^.hActiveFile := CAA.gc_hINVALID;
				close(xExecute:=FALSE);
				mxClose := 0;
			END_IF
	END_CASE
ELSE
	CASE mxRot OF
		0: // Rename
			mv(xExecute:=TRUE, sFileNameOld:=source, sFileNameNew:=dest);
			IF mv.xDone OR mv.xError THEN
				mv(xExecute:=FALSE);
				mxRot := 10;
			END_IF
		10: // Open
			open(xExecute:=TRUE, sFileName:=source, eFileMode:=FILE.MODE.MWRITE);
			IF open.xDone OR open.xError THEN
				IF open.xDone THEN
					THIS^.hActiveFile := open.hFile;
					szFilesize := 0;
					mxRot := 0;
					Rotate := TRUE;
				END_IF
				open(xExecute:=FALSE);
			END_IF
	END_CASE
	
END_IF
END_METHOD

(* Transformation file naming method.
 
 default_name will be ``sFullFilename.#``*)
METHOD PROTECTED RotationFilename : CAA.FILENAME
VAR_INPUT
	default_name	: CAA.FILENAME;
END_VAR
RotationFilename := default_name;
END_METHOD

(* Determine if we should rollover for this message. This needs to return in one call.
 This method needs to look at the next message to be written to determine if rollover should occur.*)
METHOD PROTECTED ShouldRollover : BOOL
VAR
	diLen : DINT;
	itfElementPeek : COL.IElement;
	itfSyslogMsgElementPeek : ISyslogMsgElement;
	msg : SyslogItfs.SYSLOG_MSG;
END_VAR
// Peek into the queue and see if 
IF queue.Peek(itfElement => itfElementPeek) = COL.COLLECTION_ERROR.NO_ERROR THEN
	IF __QUERYINTERFACE(itfElementPeek, itfSyslogMsgElementPeek) THEN
		msg := itfSyslogMsgElementPeek.SyslogMsgValue;
		// Add one because we append a newline
		diLen := Stu.StrLenA(ADR(msg)) + 1;
		ShouldRollover := DINT_TO___UXINT(diLen) + THIS^.szFilesize > THIS^.szMaxFilesize;
	END_IF
END_IF
END_METHOD

END_FUNCTION_BLOCK

// Handlers/SyslogRotatingFileHandlerBase
FUNCTION_BLOCK SyslogRotatingFileHandlerBase EXTENDS SyslogFileHandler
VAR_INPUT
END_VAR
VAR_OUTPUT
END_VAR
VAR
END_VAR

(* Run the handler base code*)
METHOD Run : BOOL
IF NOT xError THEN
	
	CASE mxHandler OF
		0: // Init
			IF prvFileSetup() THEN
				mxHandler := 10;
			END_IF
		10: // Process Queue
			IF ShouldRollover() AND mxQueue = 0 THEN
				DoRollover();
			ELSE
				prvProcessQueue();
				tmrFlush(IN:=TRUE);
				IF tmrFlush.Q OR xFlushNow THEN
					IF prvFlush() THEN
						tmrFlush(IN:=FALSE);
						xFlushNow := FALSE;
					END_IF
				END_IF
			END_IF
			
		20: // Reset?
			mxHandler := 0;
	END_CASE
	
END_IF
END_METHOD

END_FUNCTION_BLOCK

// Handlers/SyslogUdpHandler
{attribute 'no_assign'}
FUNCTION_BLOCK SyslogUdpHandler EXTENDS SyslogHandlerBase IMPLEMENTS SyslogItfs.ISyslogHandler
VAR_INPUT
	// Adapter IP Address that packets will be sent on
	itfAdapterAddress : NBS.IIPAddress;
	// Syslog Server IP Address
	itfServerAddress : NBS.IIPAddress;
	// Syslog UDP Port
	uiPort : UINT := SyslogItfs.gc_uiSyslogUdpPort;
	// This tells the UDP_Peer block what task to run on. If not set defaults to the task this block runs on.
	itfAsyncProperty : NBS.IAsyncProperty;
END_VAR
VAR_OUTPUT
	sError : STRING(255);
END_VAR
VAR
	peer : NBS.UDP_Peer;
	uiSendPort : UINT;
	async : NBS.AsyncProperty;
	mxRun : UINT;
	xQueueBusy : BOOL;
END_VAR

METHOD PROTECTED prvInit : BOOL
VAR_INPUT
END_VAR
VAR
	pTaskDesc : POINTER TO CmpIecTask.Task_Desc2;
	hTask : CmpIecTask.RTS_IEC_HANDLE;
	eResult : CmpIecTask.RTS_IEC_RESULT;
END_VAR
IF itfAdapterAddress <> CAA.gc_hINVALID AND itfServerAddress <> CAA.gc_hINVALID THEN
	IF itfAsyncProperty = CAA.gc_hINVALID THEN
		hTask := CmpIecTask.IecTaskGetCurrent(ADR(eResult));
		IF eResult = 0 THEN
			pTaskDesc := CmpIecTask.IecTaskGetDesc(hTask);
			IF pTaskDesc <> 0 THEN
				// I can't seem to find how to query task group 
				//async.tgTaskGroup := ?
				async.anAppName:=pTaskDesc^.pApp^.szName;
				async.tnTaskName:=pTaskDesc^.pInfo^.pszName^;
				async.usiTaskPrio:=INT_TO_USINT(pTaskDesc^.pInfo^.nPriority);
				async.udiTaskInterval:=DWORD_TO_UDINT(pTaskDesc^.pInfo^.dwInterval);
				// set the async property
				itfAsyncProperty := async;
			ELSE
				xError := TRUE;
				sError := 'Unable to get Task Descrition';
			END_IF
		ELSE
			xError := TRUE;
			sError := 'Unable to get current task';
		END_IF
	END_IF
ELSE
	xError := TRUE;
	sError := 'Missing valid adapter or server address';
END_IF

prvInit := NOT xError;
END_METHOD

METHOD PROTECTED prvProcessQueue : BOOL
VAR_INPUT
END_VAR
VAR_INST
	sCurrentMsg : SyslogItfs.SYSLOG_MSG;
END_VAR
VAR
	szLength : UDINT;
	eSendError : NBS.ERROR;
END_VAR
CASE mxQueue OF
	0: // Idle
		xQueueBusy := FALSE;
		IF queue.CountElements() > 0 THEN
			xQueueBusy := TRUE;
			mxQueue := 10;
		END_IF
	10: // Get Element
		eError := queue.Poll(itfElement => THIS^.itfElement);
		IF __QUERYINTERFACE(itfElement, itfSyslogMsgElement) THEN
			sCurrentMsg := itfSyslogMsgElement.SyslogMsgValue;
		END_IF
		
		IF eError = COL.COLLECTION_ERROR.NO_ERROR THEN
			mxQueue := 20;
		ELSE
			mxQueue := 0;
		END_IF
	20: // send
		szLength := DINT_TO_UDINT(Stu.StrLenA(ADR(sCurrentMsg)));
		eSendError := peer.Send(itfIPAddress:=itfServerAddress, uiPort:=uiPort, pData:=ADR(sCurrentMsg), udiSize:=szLength);
		CASE eSendError OF
			NBS.ERROR.NO_ERROR:
				xError := FALSE;
				sError := '';
				mxQueue := 0;
				prvProcessQueue := TRUE;
			NBS.ERROR.PENDING:
				// Pending can happen if we don't have a setup peer
				mxRun := 0;
			ELSE
				xError := TRUE;
				sError := concat('peer.Send Error: ', TO_STRING(eSendError));
		END_CASE
	ELSE
		; // NOP
END_CASE
END_METHOD

METHOD PROTECTED prvSetupConnection : BOOL
VAR_INPUT
END_VAR
IF uiSendPort = 0 THEN
	uiSendPort := RandomEmpherialPort();
END_IF

peer(xEnable:=TRUE,
	itfAsyncProperty:=itfAsyncProperty,
	itfIPAddress:=itfAdapterAddress,
	uiPort:= uiSendPort);

prvSetupConnection := peer.xActive;

IF peer.xError THEN
	xError := TRUE;
	sError := concat('Peer Error: ', TO_STRING(peer.eErrorID));
	mxRun := 0;
	peer(xEnable:=FALSE);
ELSE
	xError := FALSE;
	sError := '';
END_IF
END_METHOD

(* Run the handler base code*)
METHOD Run : BOOL
peer();

CASE mxRun OF
	0: // Init
		IF prvInit() THEN
			mxRun := 10;
		END_IF
	10: // Setup Peer
		IF prvSetupConnection() THEN
			mxRun := 20;
		END_IF
	20: // Process queue
		IF prvProcessQueue() THEN
			;
		END_IF
END_CASE
END_METHOD

END_FUNCTION_BLOCK

// SafeLog/SyslogAlert
FUNCTION SyslogAlert : BOOL
VAR_INPUT
	logger : SyslogItfs.ISyslogLogger;
	msgId	: SyslogItfs.MSG_ID;
	msg	: SyslogItfs.MSG;
END_VAR
VAR
END_VAR

IF logger <> CAA.gc_hINVALID THEN
	SyslogAlert := logger.Alert(msgId, msg);
END_IF

END_FUNCTION

// SafeLog/SyslogCritical
FUNCTION SyslogCritical : BOOL
VAR_INPUT
	logger : SyslogItfs.ISyslogLogger;
	msgId	: SyslogItfs.MSG_ID;
	msg	: SyslogItfs.MSG;
END_VAR
VAR
END_VAR

IF logger <> CAA.gc_hINVALID THEN
	SyslogCritical := logger.Critical(msgId, msg);
END_IF

END_FUNCTION

// SafeLog/SyslogDebug
FUNCTION SyslogDebug : BOOL
VAR_INPUT
	logger : SyslogItfs.ISyslogLogger;
	msgId	: SyslogItfs.MSG_ID;
	msg	: SyslogItfs.MSG;
END_VAR
VAR
END_VAR

IF logger <> CAA.gc_hINVALID THEN
	SyslogDebug := logger.Debug(msgId, msg);
END_IF

END_FUNCTION

// SafeLog/SyslogEmergency
FUNCTION SyslogEmergency : BOOL
VAR_INPUT
	logger : SyslogItfs.ISyslogLogger;
	msgId	: SyslogItfs.MSG_ID;
	msg	: SyslogItfs.MSG;
END_VAR
VAR
END_VAR

IF logger <> CAA.gc_hINVALID THEN
	SyslogEmergency := logger.Emergency(msgId, msg);
END_IF

END_FUNCTION

// SafeLog/SyslogError
FUNCTION SyslogError : BOOL
VAR_INPUT
	logger : SyslogItfs.ISyslogLogger;
	msgId	: SyslogItfs.MSG_ID;
	msg	: SyslogItfs.MSG;
END_VAR
VAR
END_VAR

IF logger <> CAA.gc_hINVALID THEN
	SyslogError := logger.Error(msgId, msg);
END_IF

END_FUNCTION

// SafeLog/SyslogInfo
FUNCTION SyslogInfo : BOOL
VAR_INPUT
	logger : SyslogItfs.ISyslogLogger;
	msgId	: SyslogItfs.MSG_ID;
	msg	: SyslogItfs.MSG;
END_VAR
VAR
END_VAR

IF logger <> CAA.gc_hINVALID THEN
	SyslogInfo := logger.Information(msgId, msg);
END_IF

END_FUNCTION

// SafeLog/SyslogNotice
FUNCTION SyslogNotice : BOOL
VAR_INPUT
	logger : SyslogItfs.ISyslogLogger;
	msgId	: SyslogItfs.MSG_ID;
	msg	: SyslogItfs.MSG;
END_VAR
VAR
END_VAR

IF logger <> CAA.gc_hINVALID THEN
	SyslogNotice := logger.Notice(msgId, msg);
END_IF

END_FUNCTION

// SafeLog/SyslogWarning
FUNCTION SyslogWarning : BOOL
VAR_INPUT
	logger : SyslogItfs.ISyslogLogger;
	msgId	: SyslogItfs.MSG_ID;
	msg	: SyslogItfs.MSG;
END_VAR
VAR
END_VAR

IF logger <> CAA.gc_hINVALID THEN
	SyslogWarning := logger.Warning(msgId, msg);
END_IF

END_FUNCTION
